TYPE ST_SITP_SygnalizacjaStanu :
STRUCT
	fbUndefined								: FB_SITP_SygnalizacjaStanu_Undefined;
	fbAborting      						: FB_SITP_SygnalizacjaStanu_Aborting;
	fbAborted       						: FB_SITP_SygnalizacjaStanu_Aborted;
	fbClearing      						: FB_SITP_SygnalizacjaStanu_Clearing;
	flSTOpping      						: FB_SITP_SygnalizacjaStanu_Stopping;
	flSTOpped       						: FB_SITP_SygnalizacjaStanu_Stopped;
	fbResetting     						: FB_SITP_SygnalizacjaStanu_Resetting;
	fbIdle          						: FB_SITP_SygnalizacjaStanu_Idle;
	fbStarting      						: FB_SITP_SygnalizacjaStanu_Starting;
	fbExecute       						: FB_SITP_SygnalizacjaStanu_Execute;
	fbSuspending    						: FB_SITP_SygnalizacjaStanu_Suspending;
	fbSuspended     						: FB_SITP_SygnalizacjaStanu_Suspended;
	fbUnsuspending  						: FB_SITP_SygnalizacjaStanu_UnSuspending;
	fbHolding       						: FB_SITP_SygnalizacjaStanu_Holding;
	fbHeld          						: FB_SITP_SygnalizacjaStanu_Held;
	fbUnholding     						: FB_SITP_SygnalizacjaStanu_UnHolding;
	fbCompleting    						: FB_SITP_SygnalizacjaStanu_Completing;
	fbComplete      						: FB_SITP_SygnalizacjaStanu_Complete;
END_STRUCT
END_TYPE

(* stored: Version 1.1.0.1
   DUT ST_SITP_SygnalizacjaStanu: Id {0e29dfdf-b372-046f-04a7-78d70e4f4fcc} *)
